ABB RAPID module: g1-code.mod

MODULE MainModule
    ! --- TARGETS ---
    CONST robtarget pPickGrid_Ref := [[359.127,0,188.4615],[0,0,0.9999999,0],[0,0,0,0],[9E+09,9E+09,9E+09,9E+09,9E+09,9E+09]];
    CONST robtarget pDestGrid_Ref := [[359.127,0,188.4615],[0,0,0.9999999,0],[0,0,0,0],[9E+09,9E+09,9E+09,9E+09,9E+09,9E+09]];

    CONST robtarget P_Color_ict:=[[266.90,275.43,180.12],[9.3566E-05,-0.709263,-0.704944,0.000120329],[0,0,1,0],[9E+09,9E+09,9E+09,9E+09,9E+09,9E+09]]
    CONST robtarget pHome := [[275.9205,0.02080205,667.3802],[0.7115182,-0.1236367,0.6797782,-0.1278957],[-1,0,-1,0],[9E+09,9E+09,9E+09,9E+09,9E+09,9E+09]];

    ! --- GRID CONSTANTS ---
    CONST num GRID_ROWS := 4;
    CONST num GRID_COLS := 4;
    CONST num OFFSET_X := 40;
    CONST num OFFSET_Y := 40;

    ! --- STATISTICS ---
    VAR num count_total := 0;
    VAR num count_correct := 0;
    VAR num count_wrong := 0;
    VAR num count_empty := 0;

   ! --- MAIN PROGRAM ---
    PROC main()
        InitProgram;

        TPWrite "Place workpieces and press start switch";

        ! ==========================================
        ! @IVAN - TASK 1: Wait for Operator
        ! INSTRUCTIONS: Use 'WaitDI' to wait for the Start_Cycle signal here.
        ! ==========================================

        TPWrite "Moving to safe Home position...";
        MoveJ pHome, v200, fine, t_grijper1\WObj:=wobj0;

        ! ==========================================
        ! @SIMONA - TASK 1: The Snake Loop
        ! INSTRUCTIONS: Delete the single ProcessBlock line below.
        ! Create nested FOR loops. Calculate the X and Y offsets.
        ! pick_target := Offs(pPickGrid_Ref, x, y, 0);
        ! drop_target := Offs(pDestGrid_Ref, x, y, 0);
        ! Call ProcessBlock(pick_target, drop_target);
        ! ==========================================

        TPWrite "Processing the grid...";
        ProcessBlock pPickGrid_Ref, pDestGrid_Ref; ! <-- SIMONA: REPLACE THIS WITH YOUR LOOPS

        TPWrite "Cycle complete. Returning Home...";
        MoveJ pHome, v200, fine, t_grijper1\WObj:=wobj0;

        ShowResults;
    ENDPROC

    ! --- SUB-PROCEDURES ---

    PROC InitProgram()
        TPErase;
        count_total := 0;
        count_correct := 0;
        count_wrong := 0;
        count_empty := 0;
    ENDPROC

    PROC ProcessBlock(robtarget pick_pos, robtarget drop_pos)
        VAR robtarget approach_pick;
        VAR robtarget approach_drop;

        approach_pick := Offs(pick_pos, 0, 0, 50);
        approach_drop := Offs(drop_pos, 0, 0, 50);

        ! Approach and descend to right platform
        MoveJ approach_pick, v200, z10, t_grijper1\WObj:=wobj0;
        MoveL pick_pos, v50, fine, t_grijper1\WObj:=wobj0;

        ! ==========================================
        ! @IVAN - TASK 2: Close the Gripper
        ! ==========================================

        ! ==========================================
        ! @BEA - TASK 1: Empty Grid Check (Error Handling)
        ! INSTRUCTIONS:
        ! 1. WaitTime 1;
        ! 2. Check DIGripperClose.
        ! 3. IF empty: Increment 'count_empty', open gripper, move back to 'approach_pick', and type 'RETURN;'
        ! ==========================================

        ! If we grabbed a block, measure it
        MeasureColor;

        ! Take block to the LEFT platform
        MoveJ approach_drop, v200, z10, t_grijper1\WObj:=wobj0;
        MoveL drop_pos, v50, fine, t_grijper1\WObj:=wobj0;

        ! ==========================================
        ! @IVAN - TASK 3: Open the Gripper
        ! ==========================================

        ! Retreat safely
        MoveL approach_drop, v100, z10, t_grijper1\WObj:=wobj0;
    ENDPROC

    PROC MeasureColor()
        ! Approach sensor safely
        MoveJ Offs(P_Color_ict, 0, 0, 50), v200, z10, t_grijper1\WObj:=wobj0;
        MoveL P_Color_ict, v50, fine, t_grijper1\WObj:=wobj0;

        ! ==========================================
        ! @BEA - TASK 2: Sensor Logic
        ! ==========================================

        ! Leave sensor safely
        MoveL Offs(P_Color_ict, 0, 0, 50), v100, z10, t_grijper1\WObj:=wobj0;
    ENDPROC

    PROC ShowResults()
        TPWrite "--- BATCH QUALITY REPORT ---";
        TPWrite "Amount of objects: " \Num:=count_total;
        TPWrite "Amount of correct colors: " \Num:=count_correct;
        TPWrite "Amount of incorrect colors: " \Num:=count_wrong;
        TPWrite "Amount of missing objects: " \Num:=count_empty;
        TPWrite "----------------------------";
    ENDPROC

ENDMODULE
